(* Logix 5000 project; controller R5_CSS vendor 1 type 14 code 74 rev 19.11; software revision 19.01; part 14 of 18 *)
(* tags used below, declared in another part *)
   P302A_QI_AUTO_OS : BOOL;
   P302A_QI_MAN_OS : BOOL;
   P302B_QI_AUTO_ONS1 : BOOL;
   FireFlowAlarmFromUTL : BOOL;
   HS315A : ValveControl_TwoWay;
   HS315B : ValveControl_TwoWay;
   LC101 : LEVEL_CONTROL;   // QUENCH TOWER BASIN LIT
   LC101_LAHH_MaxTimeAlm : BOOL;
   LC302 : LEVEL_CONTROL;   // COALESCER OIL CHAMBER LEVEL CONTROL
   LC303A : LEVEL_CONTROL;   // AQUEOUS PHASE OF PRIMARY SETTLER
   MV301 : ValveControl_TwoWay;
   ONE_SHOT : BOOL[32];
   ONE_SHOT_P303B : BOOL;
   P101B : PUMP_CONTROL;
   P302A : PUMP_CONTROL;
   P302A_PumpOut : BOOL;
   P302A_QI_AUTO_ONS1 : BOOL;
   P302A_QI_MAN_ONS1 : BOOL;
   P302B : PUMP_CONTROL;
   P302B_PumpOut : BOOL;
   P302B_QI_MAN_ONS1 : BOOL;
   P303A : PUMP_CONTROL;
   P303A_QI_AUTO_OS : BOOL;
   P303A_QI_MAN_OS : BOOL;
   P303B : PUMP_CONTROL;
   P303B_QI_AUTO_OS : BOOL;
   P303B_QI_MAN_OS : BOOL;
   TC319 : TEMP_CONTROL;   // COALESCER OIL CHAMBER PROCESS TEMPERATURE CONTROL
   TC321A : TEMP_CONTROL;   // COALESCER OIL CHAMBER TRANSFER PUMP A TEMPERATURE TRANSMITTER
   TC321B : TEMP_CONTROL;   // COALESCER OIL CHAMBER TRANSFER PUMP B TEMPERATURE TRANSMITTER
   TIMER : TIMER[50];   // HX A TIMER FOR START
(* MainProgram, continued *)

ROUTINE Pump302A_OilProductPump   (* ladder *)
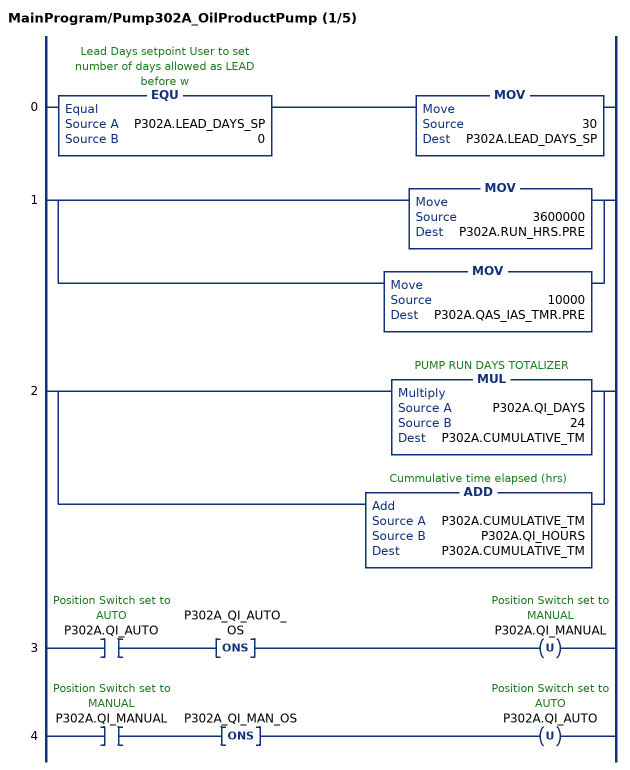
   0: EQU(P302A.LEAD_DAYS_SP,0)MOV(30,P302A.LEAD_DAYS_SP);
   1: [MOV(3600000,P302A.RUN_HRS.PRE) ,MOV(10000,P302A.QAS_IAS_TMR.PRE) ];
   2: [MUL(P302A.QI_DAYS,24,P302A.CUMULATIVE_TM) ,ADD(P302A.CUMULATIVE_TM,P302A.QI_HOURS,P302A.CUMULATIVE_TM) ];
   3: XIC(P302A.QI_AUTO)ONS(P302A_QI_AUTO_OS)OTU(P302A.QI_MANUAL);
   4: XIC(P302A.QI_MANUAL)ONS(P302A_QI_MAN_OS)OTU(P302A.QI_AUTO);
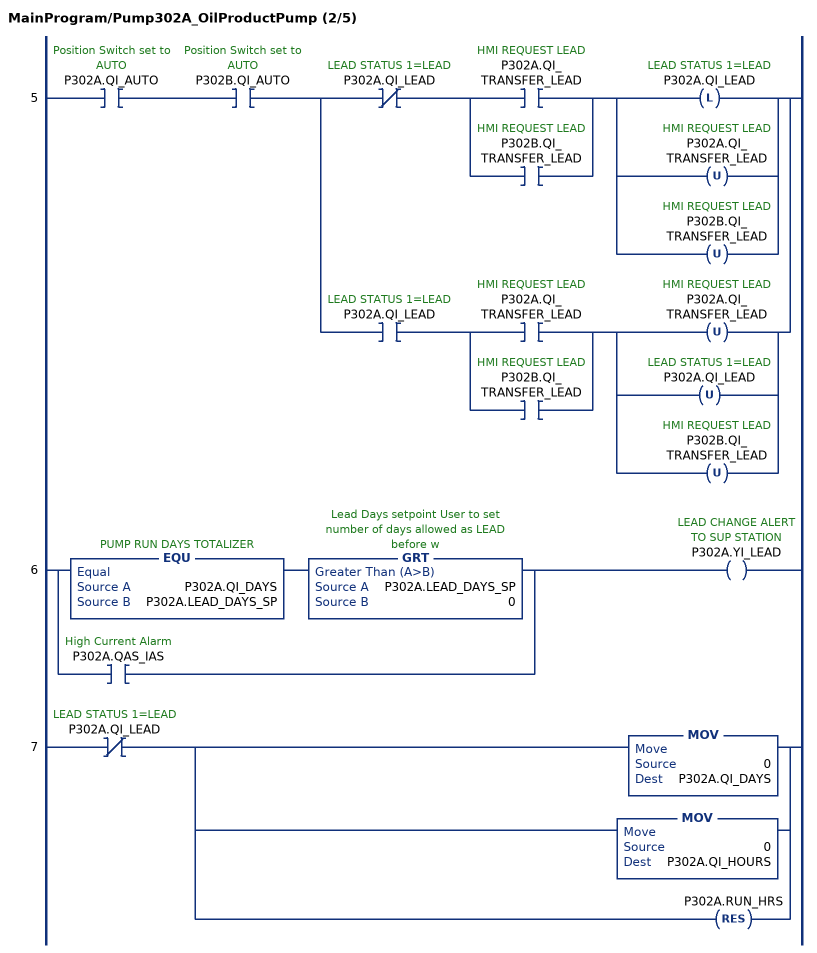
   5: XIC(P302A.QI_AUTO)XIC(P302B.QI_AUTO)[XIO(P302A.QI_LEAD) [XIC(P302A.QI_TRANSFER_LEAD) ,XIC(P302B.QI_TRANSFER_LEAD) ] [OTL(P302A.QI_LEAD) ,OTU(P302A.QI_TRANSFER_LEAD) ,OTU(P302B.QI_TRANSFER_LEAD) ] ,XIC(P302A.QI_LEAD) [XIC(P302A.QI_TRANSFER_LEAD) ,XIC(P302B.QI_TRANSFER_LEAD) ] [OTU(P302A.QI_TRANSFER_LEAD) ,OTU(P302A.QI_LEAD) ,OTU(P302B.QI_TRANSFER_LEAD) ] ];
   6: [EQU(P302A.QI_DAYS,P302A.LEAD_DAYS_SP) GRT(P302A.LEAD_DAYS_SP,0) ,XIC(P302A.QAS_IAS) ]OTE(P302A.YI_LEAD);
   7: XIO(P302A.QI_LEAD)[MOV(0,P302A.QI_DAYS) ,MOV(0,P302A.QI_HOURS) ,RES(P302A.RUN_HRS) ];
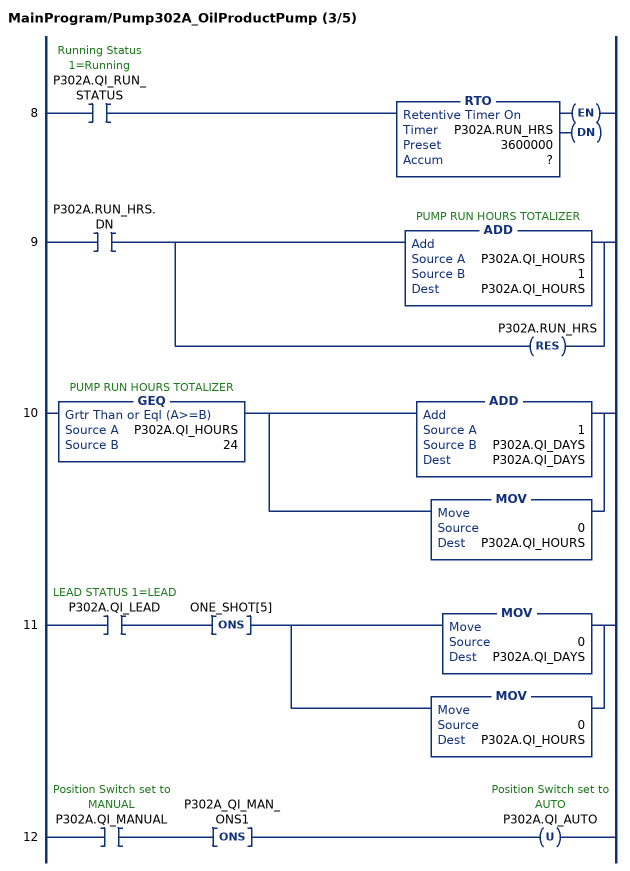
   8: XIC(P302A.QI_RUN_STATUS)RTO(P302A.RUN_HRS,?,?);
   9: XIC(P302A.RUN_HRS.DN)[ADD(P302A.QI_HOURS,1,P302A.QI_HOURS) ,RES(P302A.RUN_HRS) ];
   10: GEQ(P302A.QI_HOURS,24)[ADD(1,P302A.QI_DAYS,P302A.QI_DAYS) ,MOV(0,P302A.QI_HOURS) ];
   11: XIC(P302A.QI_LEAD)ONS(ONE_SHOT[5])[MOV(0,P302A.QI_DAYS) ,MOV(0,P302A.QI_HOURS) ];
   12: XIC(P302A.QI_MANUAL)ONS(P302A_QI_MAN_ONS1)OTU(P302A.QI_AUTO);
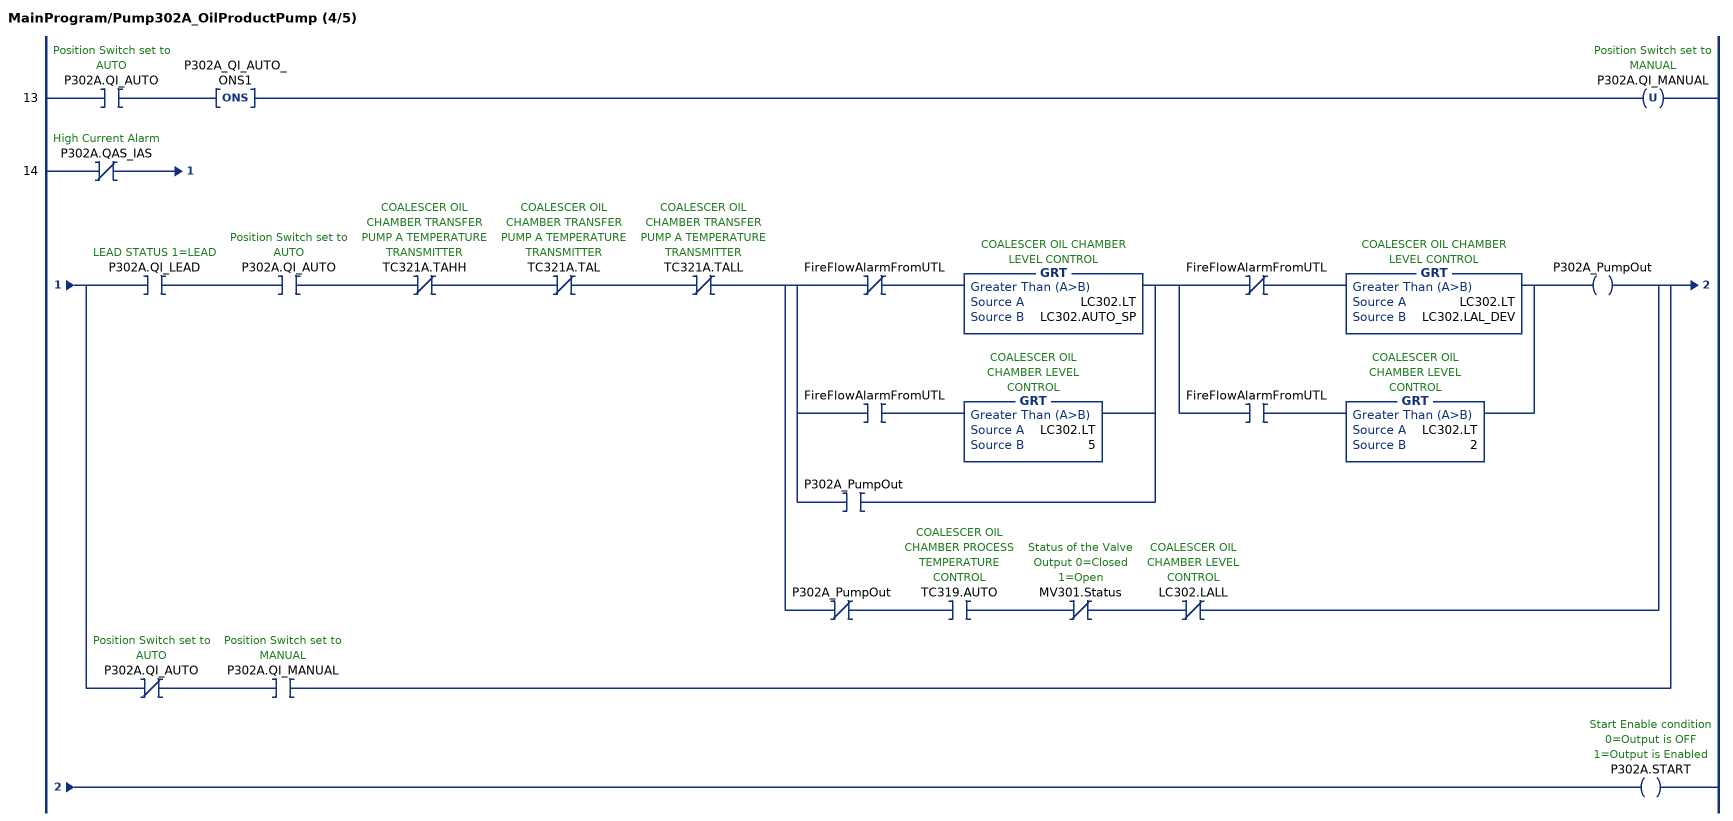
   13: XIC(P302A.QI_AUTO)ONS(P302A_QI_AUTO_ONS1)OTU(P302A.QI_MANUAL);
   14: XIO(P302A.QAS_IAS)[XIC(P302A.QI_LEAD) XIC(P302A.QI_AUTO) XIO(TC321A.TAHH) XIO(TC321A.TAL) XIO(TC321A.TALL) [[[XIO(FireFlowAlarmFromUTL) GRT(LC302.LT,LC302.AUTO_SP) ,XIC(FireFlowAlarmFromUTL) GRT(LC302.LT,5) ] ,XIC(P302A_PumpOut) ] [XIO(FireFlowAlarmFromUTL) GRT(LC302.LT,LC302.LAL_DEV) ,XIC(FireFlowAlarmFromUTL) GRT(LC302.LT,2) ] OTE(P302A_PumpOut) ,XIO(P302A_PumpOut) XIC(TC319.AUTO) XIO(MV301.Status) XIO(LC302.LALL) ] ,XIO(P302A.QI_AUTO) XIC(P302A.QI_MANUAL) ]OTE(P302A.START);
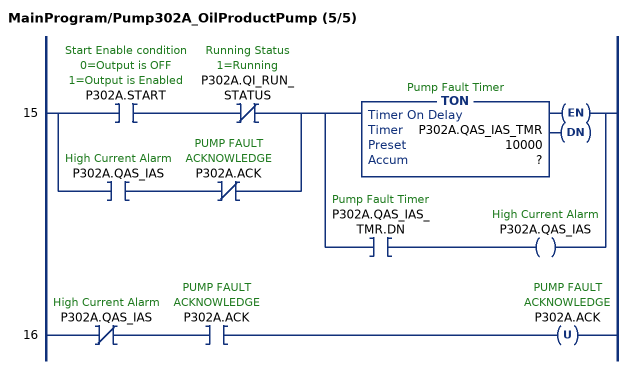
   15: [XIC(P302A.START) XIO(P302A.QI_RUN_STATUS) ,XIC(P302A.QAS_IAS) XIO(P302A.ACK) ][TON(P302A.QAS_IAS_TMR,?,?) ,XIC(P302A.QAS_IAS_TMR.DN) OTE(P302A.QAS_IAS) ];
   16: XIO(P302A.QAS_IAS)XIC(P302A.ACK)OTU(P302A.ACK);
END_ROUTINE

ROUTINE Pump302B_OilProductPump   (* ladder *)
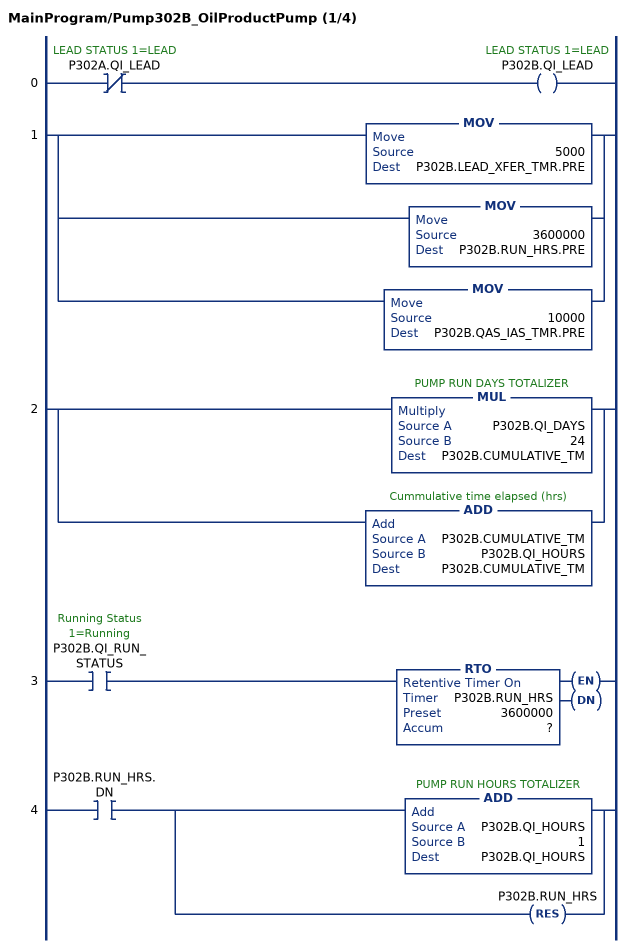
   0: XIO(P302A.QI_LEAD)OTE(P302B.QI_LEAD);
   1: [MOV(5000,P302B.LEAD_XFER_TMR.PRE) ,MOV(3600000,P302B.RUN_HRS.PRE) ,MOV(10000,P302B.QAS_IAS_TMR.PRE) ];
   2: [MUL(P302B.QI_DAYS,24,P302B.CUMULATIVE_TM) ,ADD(P302B.CUMULATIVE_TM,P302B.QI_HOURS,P302B.CUMULATIVE_TM) ];
   3: XIC(P302B.QI_RUN_STATUS)RTO(P302B.RUN_HRS,?,?);
   4: XIC(P302B.RUN_HRS.DN)[ADD(P302B.QI_HOURS,1,P302B.QI_HOURS) ,RES(P302B.RUN_HRS) ];
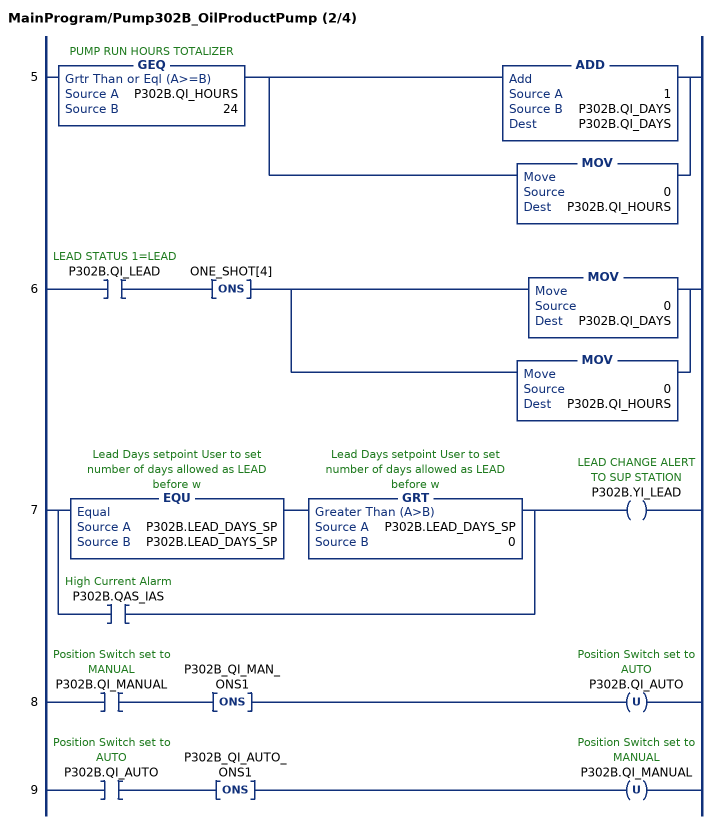
   5: GEQ(P302B.QI_HOURS,24)[ADD(1,P302B.QI_DAYS,P302B.QI_DAYS) ,MOV(0,P302B.QI_HOURS) ];
   6: XIC(P302B.QI_LEAD)ONS(ONE_SHOT[4])[MOV(0,P302B.QI_DAYS) ,MOV(0,P302B.QI_HOURS) ];
   7: [EQU(P302B.LEAD_DAYS_SP,P302B.LEAD_DAYS_SP) GRT(P302B.LEAD_DAYS_SP,0) ,XIC(P302B.QAS_IAS) ]OTE(P302B.YI_LEAD);
   8: XIC(P302B.QI_MANUAL)ONS(P302B_QI_MAN_ONS1)OTU(P302B.QI_AUTO);
   9: XIC(P302B.QI_AUTO)ONS(P302B_QI_AUTO_ONS1)OTU(P302B.QI_MANUAL);
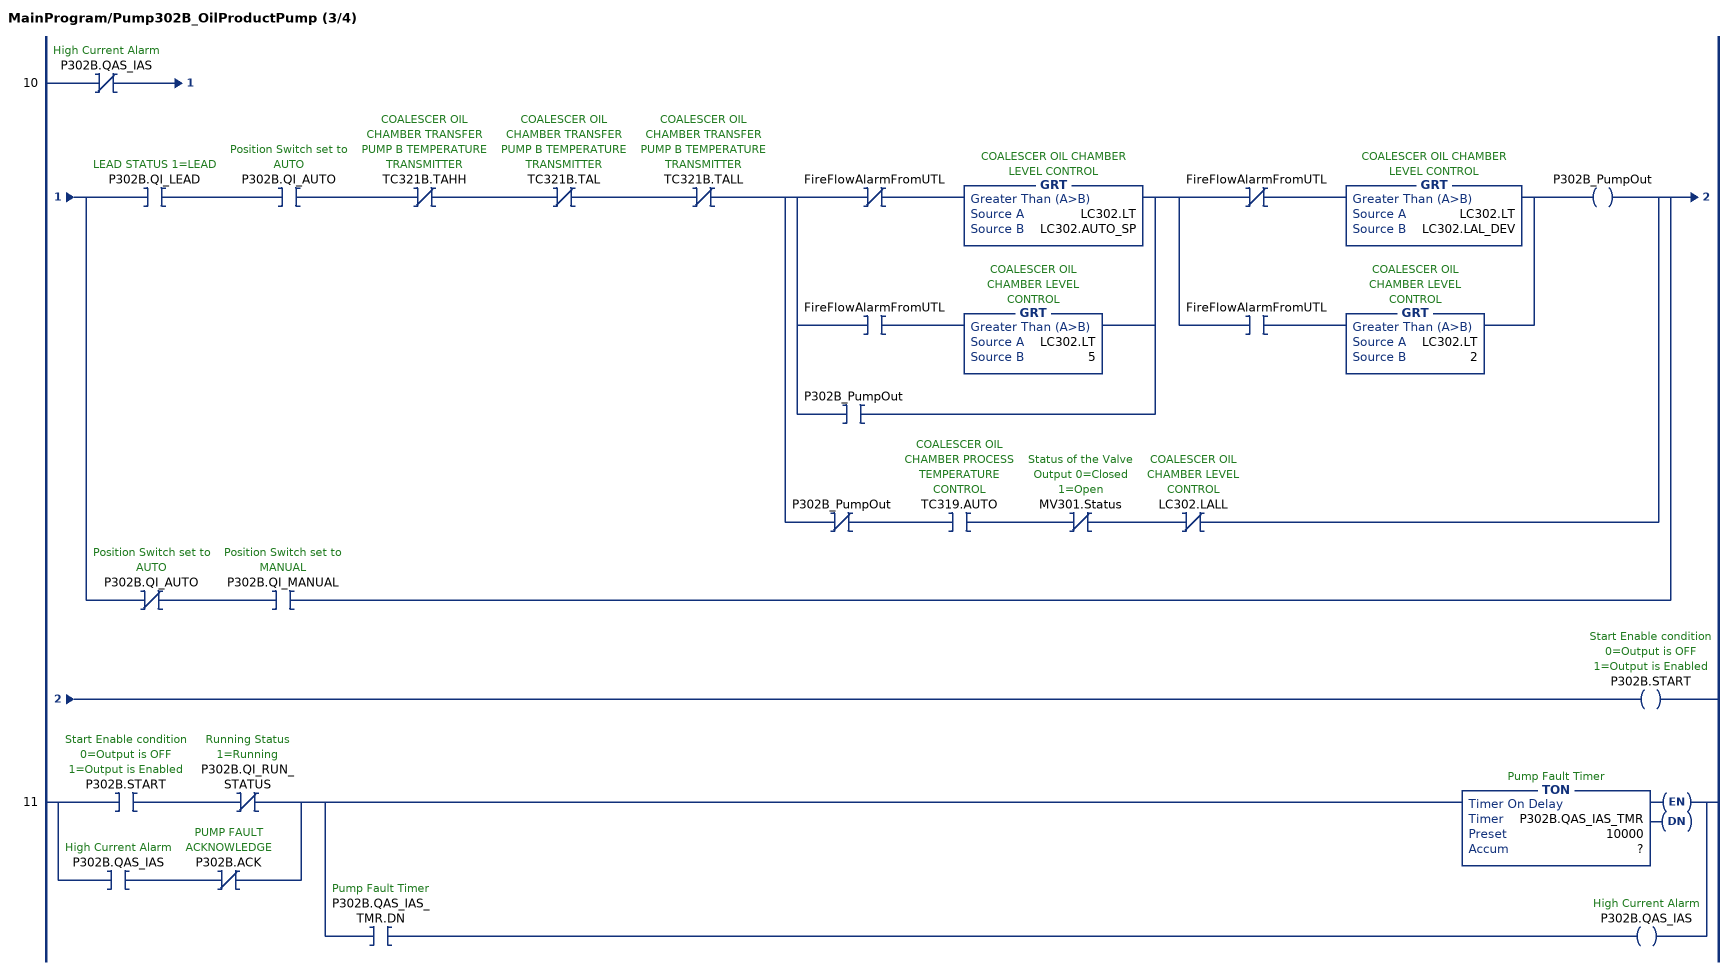
   10: XIO(P302B.QAS_IAS)[XIC(P302B.QI_LEAD) XIC(P302B.QI_AUTO) XIO(TC321B.TAHH) XIO(TC321B.TAL) XIO(TC321B.TALL) [[[XIO(FireFlowAlarmFromUTL) GRT(LC302.LT,LC302.AUTO_SP) ,XIC(FireFlowAlarmFromUTL) GRT(LC302.LT,5) ] ,XIC(P302B_PumpOut) ] [XIO(FireFlowAlarmFromUTL) GRT(LC302.LT,LC302.LAL_DEV) ,XIC(FireFlowAlarmFromUTL) GRT(LC302.LT,2) ] OTE(P302B_PumpOut) ,XIO(P302B_PumpOut) XIC(TC319.AUTO) XIO(MV301.Status) XIO(LC302.LALL) ] ,XIO(P302B.QI_AUTO) XIC(P302B.QI_MANUAL) ]OTE(P302B.START);
   11: [XIC(P302B.START) XIO(P302B.QI_RUN_STATUS) ,XIC(P302B.QAS_IAS) XIO(P302B.ACK) ][TON(P302B.QAS_IAS_TMR,?,?) ,XIC(P302B.QAS_IAS_TMR.DN) OTE(P302B.QAS_IAS) ];
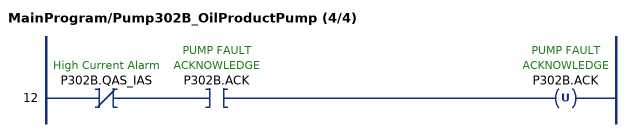
   12: XIO(P302B.QAS_IAS)XIC(P302B.ACK)OTU(P302B.ACK);
END_ROUTINE

ROUTINE Pump303A_QuenchWaterPump   (* ladder *)
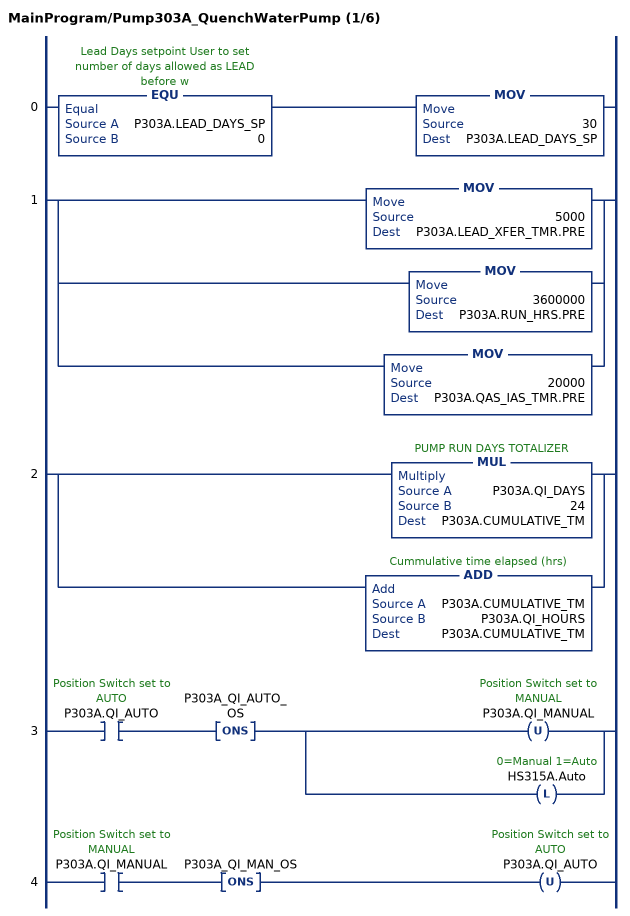
   0: EQU(P303A.LEAD_DAYS_SP,0)MOV(30,P303A.LEAD_DAYS_SP);
   1: [MOV(5000,P303A.LEAD_XFER_TMR.PRE) ,MOV(3600000,P303A.RUN_HRS.PRE) ,MOV(20000,P303A.QAS_IAS_TMR.PRE) ];
   2: [MUL(P303A.QI_DAYS,24,P303A.CUMULATIVE_TM) ,ADD(P303A.CUMULATIVE_TM,P303A.QI_HOURS,P303A.CUMULATIVE_TM) ];
   3: XIC(P303A.QI_AUTO)ONS(P303A_QI_AUTO_OS)[OTU(P303A.QI_MANUAL) ,OTL(HS315A.Auto) ];
   4: XIC(P303A.QI_MANUAL)ONS(P303A_QI_MAN_OS)OTU(P303A.QI_AUTO);
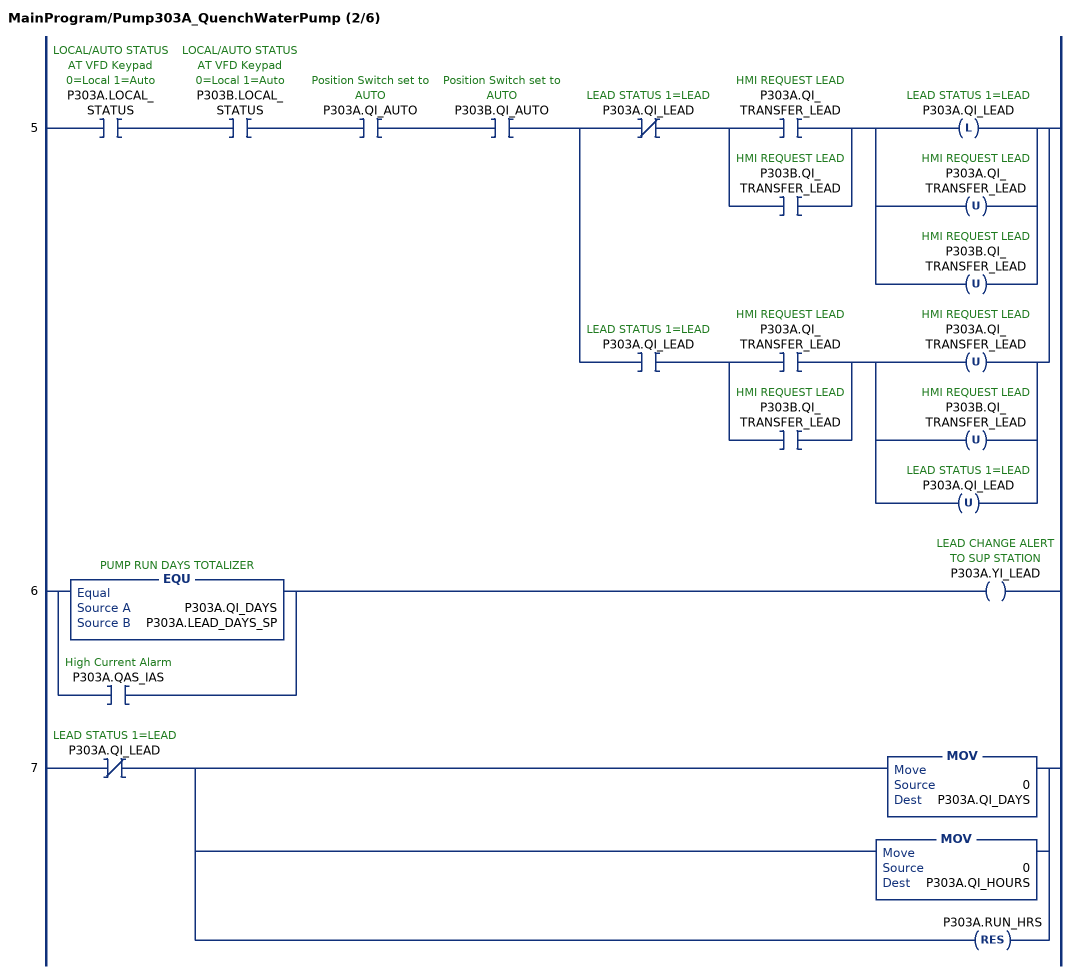
   5: XIC(P303A.LOCAL_STATUS)XIC(P303B.LOCAL_STATUS)XIC(P303A.QI_AUTO)XIC(P303B.QI_AUTO)[XIO(P303A.QI_LEAD) [XIC(P303A.QI_TRANSFER_LEAD) ,XIC(P303B.QI_TRANSFER_LEAD) ] [OTL(P303A.QI_LEAD) ,OTU(P303A.QI_TRANSFER_LEAD) ,OTU(P303B.QI_TRANSFER_LEAD) ] ,XIC(P303A.QI_LEAD) [XIC(P303A.QI_TRANSFER_LEAD) ,XIC(P303B.QI_TRANSFER_LEAD) ] [OTU(P303A.QI_TRANSFER_LEAD) ,OTU(P303B.QI_TRANSFER_LEAD) ,OTU(P303A.QI_LEAD) ] ];
   6: [EQU(P303A.QI_DAYS,P303A.LEAD_DAYS_SP) ,XIC(P303A.QAS_IAS) ]OTE(P303A.YI_LEAD);
   7: XIO(P303A.QI_LEAD)[MOV(0,P303A.QI_DAYS) ,MOV(0,P303A.QI_HOURS) ,RES(P303A.RUN_HRS) ];
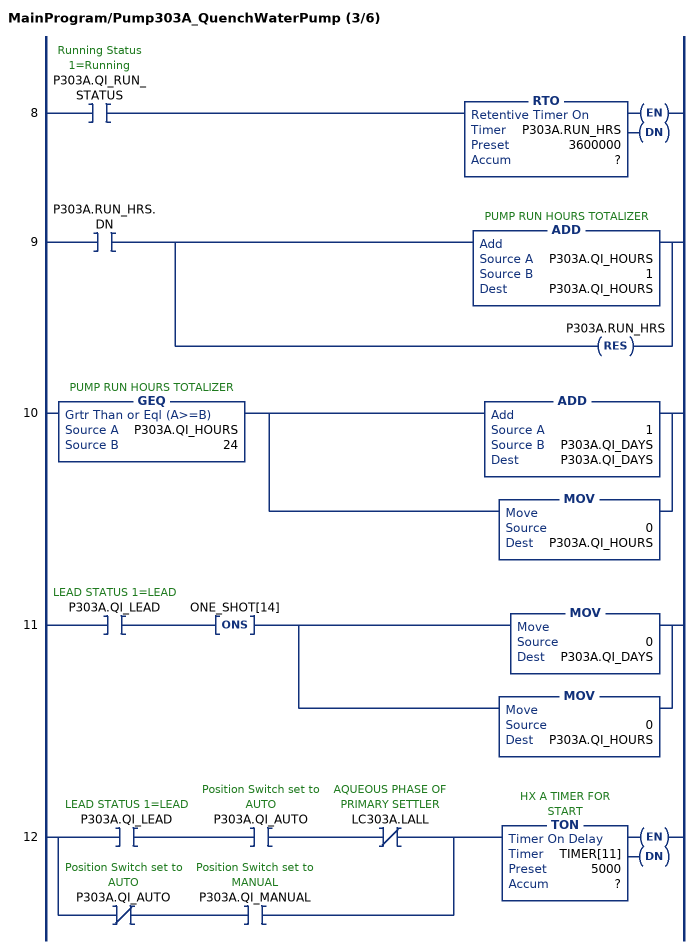
   8: XIC(P303A.QI_RUN_STATUS)RTO(P303A.RUN_HRS,?,?);
   9: XIC(P303A.RUN_HRS.DN)[ADD(P303A.QI_HOURS,1,P303A.QI_HOURS) ,RES(P303A.RUN_HRS) ];
   10: GEQ(P303A.QI_HOURS,24)[ADD(1,P303A.QI_DAYS,P303A.QI_DAYS) ,MOV(0,P303A.QI_HOURS) ];
   11: XIC(P303A.QI_LEAD)ONS(ONE_SHOT[14])[MOV(0,P303A.QI_DAYS) ,MOV(0,P303A.QI_HOURS) ];
   12: [XIC(P303A.QI_LEAD) XIC(P303A.QI_AUTO) XIO(LC303A.LALL) ,XIO(P303A.QI_AUTO) XIC(P303A.QI_MANUAL) ]TON(TIMER[11],?,?);
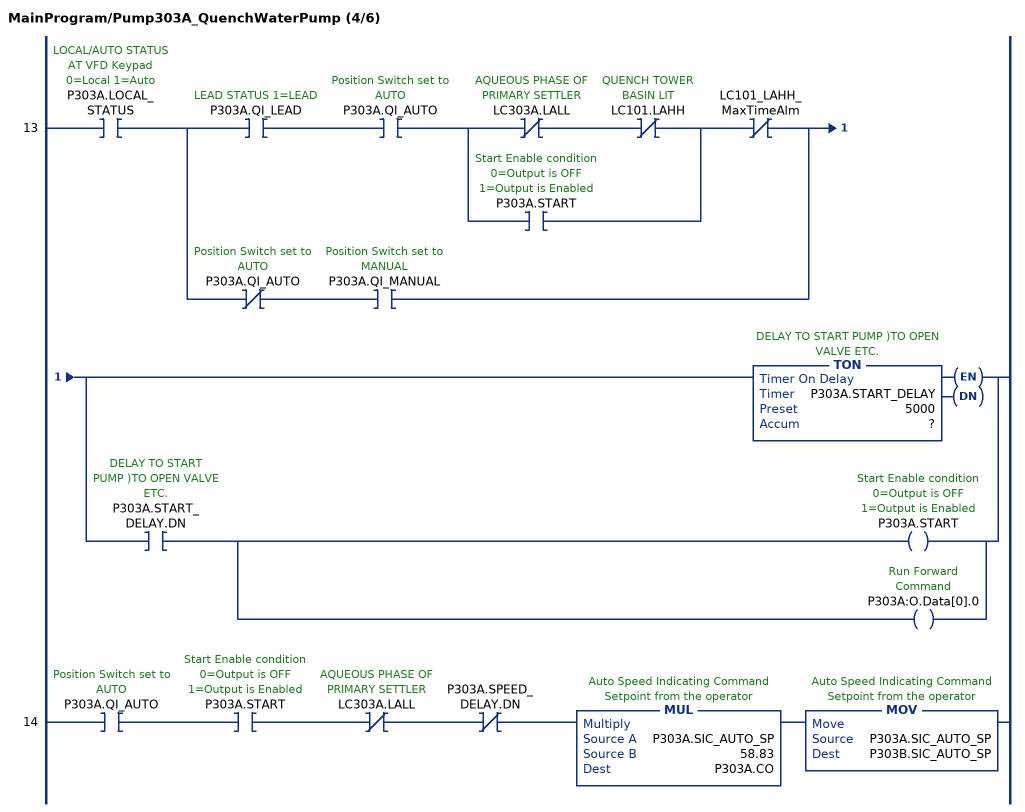
   13: XIC(P303A.LOCAL_STATUS)[XIC(P303A.QI_LEAD) XIC(P303A.QI_AUTO) [XIO(LC303A.LALL) XIO(LC101.LAHH) ,XIC(P303A.START) ] XIO(LC101_LAHH_MaxTimeAlm) ,XIO(P303A.QI_AUTO) XIC(P303A.QI_MANUAL) ][TON(P303A.START_DELAY,?,?) ,XIC(P303A.START_DELAY.DN) [OTE(P303A.START) ,OTE(P303A:O.Data[0].0) ] ];
   14: XIC(P303A.QI_AUTO)XIC(P303A.START)XIO(LC303A.LALL)XIO(P303A.SPEED_DELAY.DN)MUL(P303A.SIC_AUTO_SP,58.83,P303A.CO)MOV(P303A.SIC_AUTO_SP,P303B.SIC_AUTO_SP);
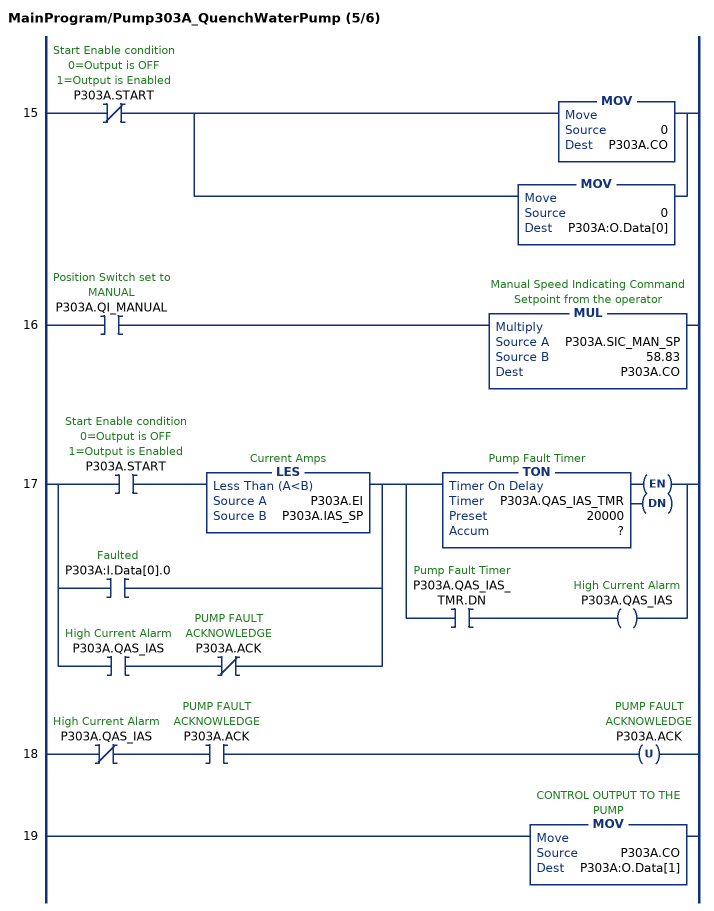
   15: XIO(P303A.START)[MOV(0,P303A.CO) ,MOV(0,P303A:O.Data[0]) ];
   16: XIC(P303A.QI_MANUAL)MUL(P303A.SIC_MAN_SP,58.83,P303A.CO);
   17: [XIC(P303A.START) LES(P303A.EI,P303A.IAS_SP) ,XIC(P303A:I.Data[0].0) ,XIC(P303A.QAS_IAS) XIO(P303A.ACK) ][TON(P303A.QAS_IAS_TMR,?,?) ,XIC(P303A.QAS_IAS_TMR.DN) OTE(P303A.QAS_IAS) ];
   18: XIO(P303A.QAS_IAS)XIC(P303A.ACK)OTU(P303A.ACK);
   19: MOV(P303A.CO,P303A:O.Data[1]);
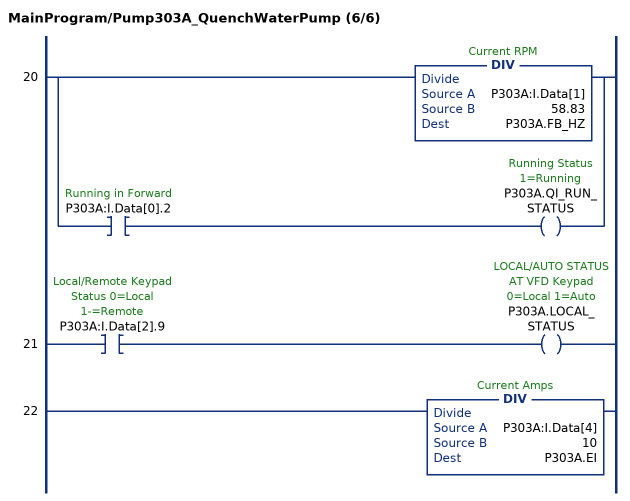
   20: [DIV(P303A:I.Data[1],58.83,P303A.FB_HZ) ,XIC(P303A:I.Data[0].2) OTE(P303A.QI_RUN_STATUS) ];
   21: XIC(P303A:I.Data[2].9)OTE(P303A.LOCAL_STATUS);
   22: DIV(P303A:I.Data[4],10,P303A.EI);
END_ROUTINE

ROUTINE Pump303B_QuenchWaterPump   (* ladder *)
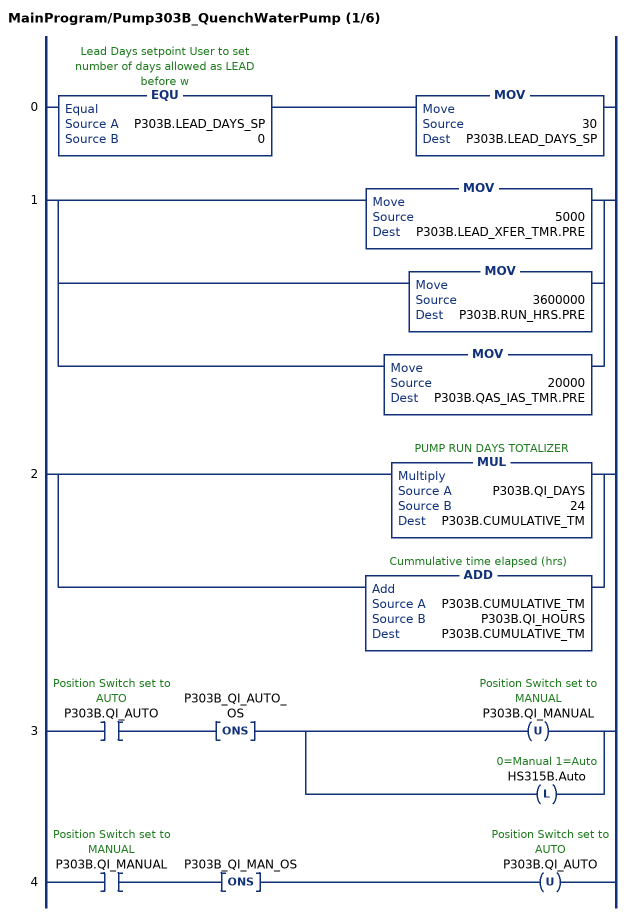
   0: EQU(P303B.LEAD_DAYS_SP,0)MOV(30,P303B.LEAD_DAYS_SP);
   1: [MOV(5000,P303B.LEAD_XFER_TMR.PRE) ,MOV(3600000,P303B.RUN_HRS.PRE) ,MOV(20000,P303B.QAS_IAS_TMR.PRE) ];
   2: [MUL(P303B.QI_DAYS,24,P303B.CUMULATIVE_TM) ,ADD(P303B.CUMULATIVE_TM,P303B.QI_HOURS,P303B.CUMULATIVE_TM) ];
   3: XIC(P303B.QI_AUTO)ONS(P303B_QI_AUTO_OS)[OTU(P303B.QI_MANUAL) ,OTL(HS315B.Auto) ];
   4: XIC(P303B.QI_MANUAL)ONS(P303B_QI_MAN_OS)OTU(P303B.QI_AUTO);
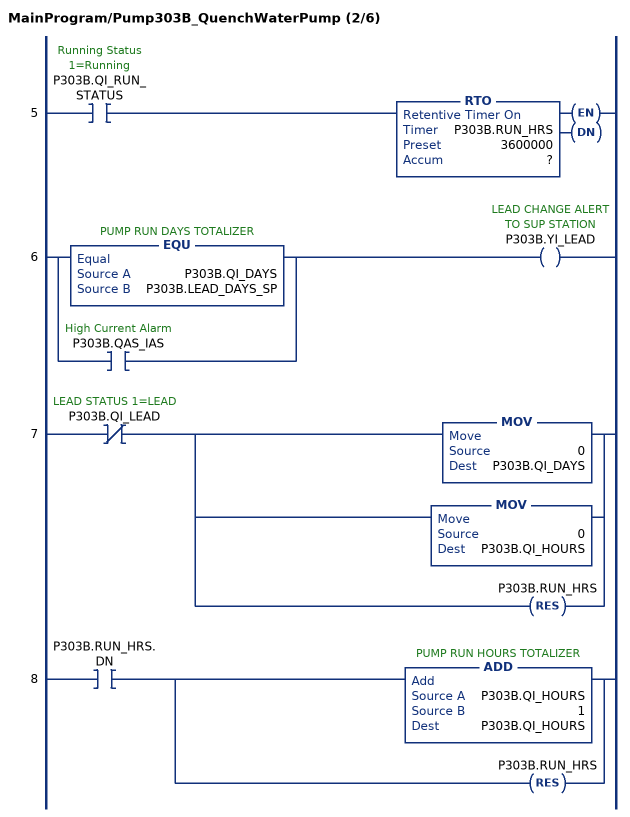
   5: XIC(P303B.QI_RUN_STATUS)RTO(P303B.RUN_HRS,?,?);
   6: [EQU(P303B.QI_DAYS,P303B.LEAD_DAYS_SP) ,XIC(P303B.QAS_IAS) ]OTE(P303B.YI_LEAD);
   7: XIO(P303B.QI_LEAD)[MOV(0,P303B.QI_DAYS) ,MOV(0,P303B.QI_HOURS) ,RES(P303B.RUN_HRS) ];
   8: XIC(P303B.RUN_HRS.DN)[ADD(P303B.QI_HOURS,1,P303B.QI_HOURS) ,RES(P303B.RUN_HRS) ];
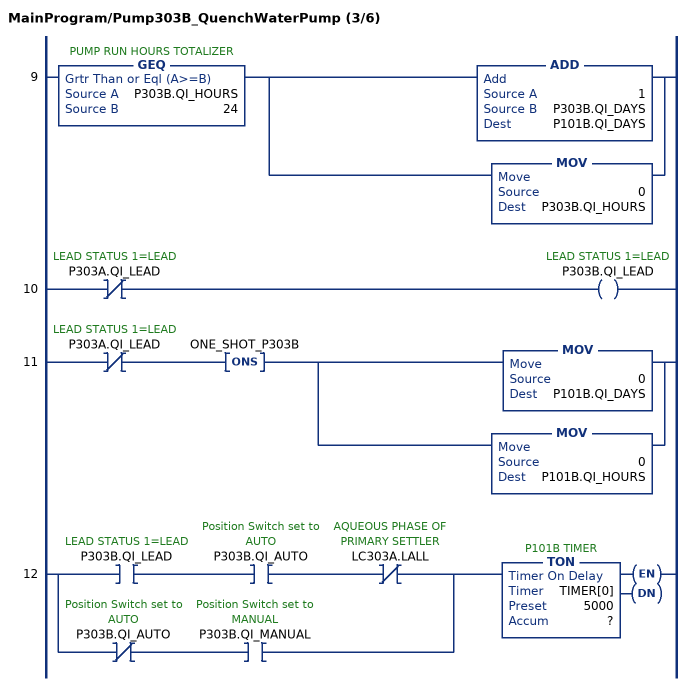
   9: GEQ(P303B.QI_HOURS,24)[ADD(1,P303B.QI_DAYS,P101B.QI_DAYS) ,MOV(0,P303B.QI_HOURS) ];
   10: XIO(P303A.QI_LEAD)OTE(P303B.QI_LEAD);
   11: XIO(P303A.QI_LEAD)ONS(ONE_SHOT_P303B)[MOV(0,P101B.QI_DAYS) ,MOV(0,P101B.QI_HOURS) ];
   12: [XIC(P303B.QI_LEAD) XIC(P303B.QI_AUTO) XIO(LC303A.LALL) ,XIO(P303B.QI_AUTO) XIC(P303B.QI_MANUAL) ]TON(TIMER[0],?,?);
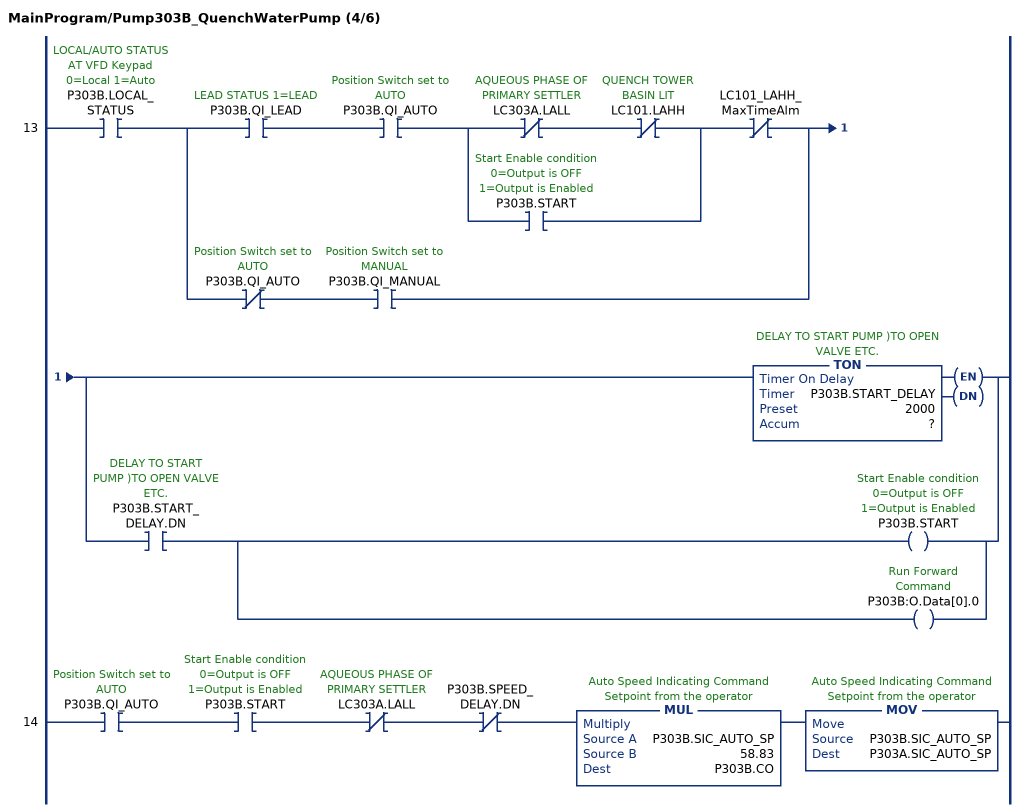
   13: XIC(P303B.LOCAL_STATUS)[XIC(P303B.QI_LEAD) XIC(P303B.QI_AUTO) [XIO(LC303A.LALL) XIO(LC101.LAHH) ,XIC(P303B.START) ] XIO(LC101_LAHH_MaxTimeAlm) ,XIO(P303B.QI_AUTO) XIC(P303B.QI_MANUAL) ][TON(P303B.START_DELAY,?,?) ,XIC(P303B.START_DELAY.DN) [OTE(P303B.START) ,OTE(P303B:O.Data[0].0) ] ];
   14: XIC(P303B.QI_AUTO)XIC(P303B.START)XIO(LC303A.LALL)XIO(P303B.SPEED_DELAY.DN)MUL(P303B.SIC_AUTO_SP,58.83,P303B.CO)MOV(P303B.SIC_AUTO_SP,P303A.SIC_AUTO_SP);
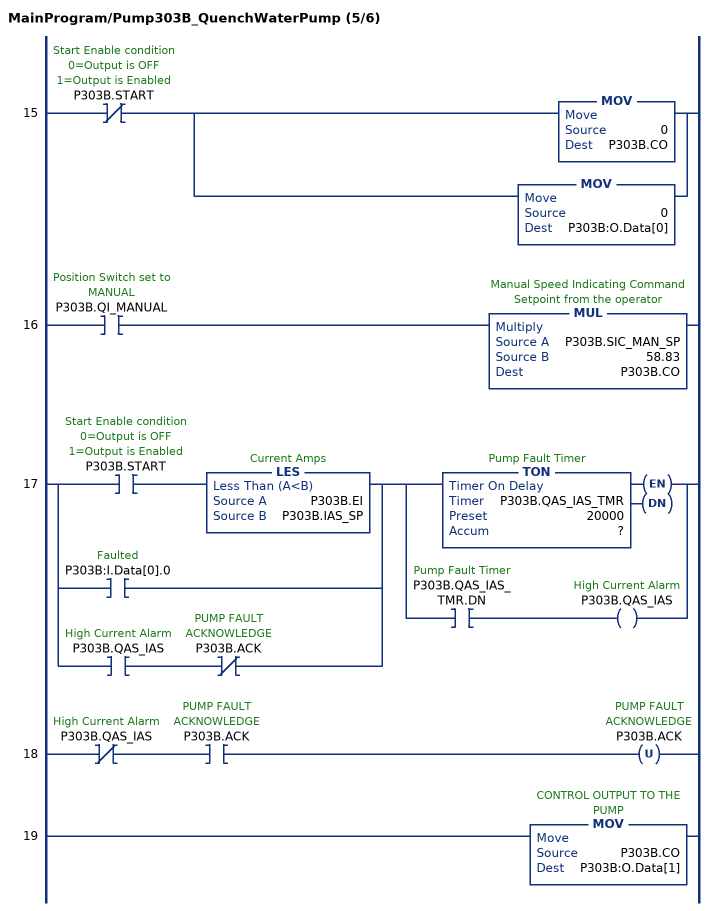
   15: XIO(P303B.START)[MOV(0,P303B.CO) ,MOV(0,P303B:O.Data[0]) ];
   16: XIC(P303B.QI_MANUAL)MUL(P303B.SIC_MAN_SP,58.83,P303B.CO);
   17: [XIC(P303B.START) LES(P303B.EI,P303B.IAS_SP) ,XIC(P303B:I.Data[0].0) ,XIC(P303B.QAS_IAS) XIO(P303B.ACK) ][TON(P303B.QAS_IAS_TMR,?,?) ,XIC(P303B.QAS_IAS_TMR.DN) OTE(P303B.QAS_IAS) ];
   18: XIO(P303B.QAS_IAS)XIC(P303B.ACK)OTU(P303B.ACK);
   19: MOV(P303B.CO,P303B:O.Data[1]);
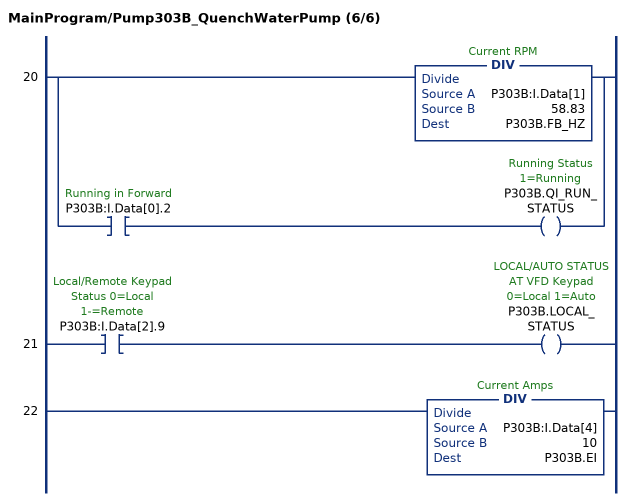
   20: [DIV(P303B:I.Data[1],58.83,P303B.FB_HZ) ,XIC(P303B:I.Data[0].2) OTE(P303B.QI_RUN_STATUS) ];
   21: XIC(P303B:I.Data[2].9)OTE(P303B.LOCAL_STATUS);
   22: DIV(P303B:I.Data[4],10,P303B.EI);
END_ROUTINE
